Yaskawa INFORM job: SKRZYNIA_4740_90_STOPNI_20BR.JBI

/JOB
//NAME SKRZYNIA_4740_90_STOPNI_20BR
///FOLDERNAME 02-SKRZYNIE_JOBS
//POS
///NPOS 536,536,0,37,0,0
///TOOL 0
///POSTYPE PULSE
///PULSE
C00000=0,-52280,40443,0,6876,0
C00001=82314,-24956,17040,59626,-27382,6248
C00002=93910,-8625,17040,59626,-43355,6248
C00003=98846,-1061,-42166,80308,-57081,-16120
C00004=100452,6057,-48127,85711,-56704,-21322
C00005=95573,33077,-33257,84645,-64023,-26851
C00006=94102,33899,-31937,85246,-63371,-26689
C00007=95573,33077,-33257,84645,-64023,-26851
C00008=94862,31071,-36438,85313,-63677,-27192
C00009=95573,33077,-33257,84645,-64023,-26851
C00010=95263,33142,-33256,84677,-63995,-26850
C00011=95263,33142,-33256,84677,-63995,-26850
C00012=94017,33843,-32133,85187,-63445,-26710
C00013=95263,33142,-33256,84677,-63995,-26850
C00014=94657,31439,-35966,85248,-63701,-27141
C00015=95263,33142,-33256,84677,-63995,-26850
C00016=95260,33144,-33256,84678,-63995,-26850
C00017=95260,33144,-33256,84678,-63995,-26850
C00018=94022,33838,-32141,85183,-63448,-26711
C00019=95260,33144,-33256,84678,-63995,-26850
C00020=94618,31343,-36117,85281,-63684,-27157
C00021=95260,33144,-33256,84678,-63995,-26850
C00022=95258,25631,32269,66559,-75499,-2416
C00023=95258,25631,32269,66559,-75499,-2416
C00024=94181,26497,33533,66410,-74896,-2191
C00025=95658,30184,39035,66708,-78559,-2356
C00026=95217,30377,39331,66881,-79841,-2558
C00027=95258,25631,32269,66559,-75499,-2416
C00028=98811,21047,-15512,99242,-81394,-20987
C00029=98811,21047,-15512,99242,-81394,-20987
C00030=97775,21639,-14693,99563,-80753,-20993
C00031=98811,21047,-15512,99242,-81394,-20987
C00032=98206,18840,-18520,99489,-81124,-21211
C00033=98811,21047,-15512,99242,-81394,-20987
C00034=97770,33535,58109,97477,-73223,-2907
C00035=97471,32489,56434,97533,-73096,-3098
C00036=96615,33295,57725,97337,-72490,-3014
C00037=97471,32489,56434,97533,-73096,-3098
C00038=97097,30483,53272,97662,-72975,-3435
C00039=97471,32489,56434,97533,-73096,-3098
C00040=98003,23984,26658,100907,-76471,-9645
C00041=97707,-10819,-23052,107304,-59718,-16318
C00042=94212,-35028,-34485,100444,-49148,-11285
C00043=48287,-44591,-17414,16172,-14532,25809
C00044=85348,-13130,13838,41209,-47455,8220
C00045=97395,20012,29210,69700,-74457,-9077
C00046=97055,28839,36684,71776,-79389,-10554
C00047=97055,28839,36684,71776,-79389,-10554
C00048=96058,29646,37897,71666,-78799,-10362
C00049=97055,28839,36684,71776,-79389,-10554
C00050=96570,26659,33451,71832,-78911,-10777
C00051=97055,28839,36684,71776,-79389,-10554
C00052=99260,22658,16753,92099,-78835,-1091
C00053=98782,22427,16945,92082,-78485,-960
C00054=98098,22870,17565,92116,-78014,-935
C00055=98782,22427,16945,92082,-78485,-960
C00056=98488,21195,15235,92147,-78307,-1085
C00057=98782,22427,16945,92082,-78485,-960
C00058=99953,7972,-32104,116782,-84999,-13620
C00059=94704,-17776,-58548,118507,-81680,-13914
C00060=60067,-64368,-72505,144806,-26050,-19168
C00061=60067,-50244,-32501,110603,-14199,-2207
C00062=63330,-26972,24478,18707,-56801,31483
C00063=95462,-31003,-33042,65414,-41305,6524
C00064=97787,-9790,-26685,81509,-54738,-4408
C00065=99864,21793,7359,80466,-76601,-6182
C00066=99753,21489,3165,89598,-79157,-3178
C00067=99071,20978,1948,89791,-78725,-3400
C00068=98206,21502,2669,89926,-78149,-3364
C00069=99071,20978,1948,89791,-78725,-3400
C00070=98727,19613,87,89895,-78511,-3524
C00071=99071,20978,1948,89791,-78725,-3400
C00072=99862,21793,7358,80466,-76600,-6182
C00073=98290,21024,6297,80683,-75539,-6194
C00074=97471,21541,7008,80756,-75007,-6115
C00075=98290,21024,6297,80683,-75539,-6194
C00076=97834,19245,3873,80814,-75197,-6333
C00077=98290,21024,6297,80683,-75539,-6194
C00078=98946,26804,31705,85784,-78857,-1423
C00079=98946,26804,31705,85784,-78857,-1423
C00080=98292,27270,32391,85749,-78414,-1361
C00081=98946,26804,31705,85784,-78857,-1423
C00082=98631,25349,29587,85839,-78632,-1590
C00083=98946,26804,31705,85784,-78857,-1423
C00084=94295,-1388,2615,87521,-55608,-1527
C00085=77022,-27457,-20499,75297,-20933,3764
///LIMIT ON
C00086=42754,-66126,12236,-1301,3231,7194
///LIMIT OFF
C00087=0,-52280,40443,0,6876,0
C00088=0,-52280,40443,0,6876,0
C00089=50509,-19000,10610,51503,-15997,-61182
C00090=50873,-17966,11417,52677,-16048,-61710
C00091=49459,-16590,12517,51258,-15158,-61190
C00092=50592,-16429,12648,53120,-15720,-61960
C00093=50873,-17966,11417,52677,-16048,-61710
C00094=50703,-18403,11066,52155,-16024,-61477
C00095=50703,-18403,11066,52155,-16024,-61477
C00096=49026,-16768,12358,50435,-14971,-60844
C00097=50653,-16371,12680,53228,-15754,-62008
C00098=50703,-18403,11066,52155,-16024,-61477
C00099=50704,-18401,11069,52157,-16021,-61478
C00100=50704,-20525,5414,58956,-14779,-64789
C00101=49025,-18889,6668,57745,-13658,-64384
C00102=50799,-18420,7036,60610,-14610,-65581
C00103=50704,-20525,5414,58956,-14779,-64789
C00104=51005,-17995,11387,52847,-16122,-61778
C00105=51005,-17995,11387,52847,-16122,-61778
C00106=49564,-16598,12501,51417,-15218,-61257
C00107=50954,-16306,12737,53719,-15902,-62212
C00108=51005,-17995,11387,52847,-16122,-61778
C00109=51030,-17981,11395,52891,-16138,-61796
C00110=51030,-17981,11395,52891,-16138,-61796
C00111=49401,-16396,12662,51265,-15114,-61201
C00112=50908,-16047,12947,53789,-15850,-62250
C00113=51030,-17981,11395,52891,-16138,-61796
C00114=50945,-18019,11363,52741,-16103,-61737
C00115=50945,-16980,14081,49884,-16761,-60338
C00116=49117,-15186,15539,47848,-15653,-59576
C00117=50939,-14679,15960,50992,-16487,-60881
C00118=50945,-18019,11363,52741,-16103,-61737
C00119=50945,-18019,11363,52741,-16103,-61737
C00120=50945,-18556,9943,54337,-15776,-62517
C00121=48967,-16606,11493,52445,-14510,-61829
C00122=51083,-15952,12027,56053,-15559,-63336
C00123=50945,-18556,9943,54337,-15776,-62517
C00124=50945,-18019,11363,52741,-16103,-61737
C00125=51350,-15183,18375,46705,-17991,-58719
C00126=49319,-13187,20053,44263,-16830,-57796
C00127=51236,-12618,20544,47529,-17647,-59142
C00128=51350,-15183,18375,46705,-17991,-58719
C00129=50028,-23690,-6096,22921,-31075,-54538
C00130=50670,-23735,-6923,24003,-30760,-55076
C00131=48518,-21492,-5254,21861,-29696,-54082
C00132=50138,-21068,-4928,23831,-30039,-55022
C00133=50670,-23735,-6923,24003,-30760,-55076
C00134=49763,-24225,-29961,22080,-30065,-59113
C00135=49763,-24225,-29961,22080,-30065,-59113
C00136=47727,-21550,-27874,20313,-29013,-58119
C00137=49271,-21042,-27466,22016,-29310,-59069
C00138=49763,-24225,-29961,22080,-30065,-59113
C00139=50713,-12366,-58367,41124,-17813,-74400
C00140=50713,-12366,-58367,41124,-17813,-74400
C00141=48934,-9522,-55687,39981,-16902,-73526
C00142=50242,-8975,-55157,41389,-17374,-74448
C00143=50713,-12366,-58367,41124,-17813,-74400
C00144=50713,-12366,-58367,41124,-17813,-74400
C00145=50713,-12366,-58367,41124,-17813,-74400
C00146=48934,-9522,-55687,39981,-16902,-73526
C00147=50242,-8975,-55157,41389,-17374,-74448
C00148=50713,-12366,-58367,41124,-17813,-74400
C00149=49763,-25421,-36239,24565,-26935,-60445
C00150=43547,-31626,-19626,5157,-49140,-52118
C00151=40154,-51179,-915,24203,-8234,-36524
C00152=0,-52280,40443,0,6876,0
C00153=0,-52280,40443,0,6876,0
C00154=2117,-50103,-33543,4117,45077,-85249
C00155=-26439,-48928,-33543,4117,-52362,-85249
C00156=-1453,-29933,-32011,46693,-66666,-90474
C00157=24798,-19255,-10490,69050,-85424,-90395
C00158=18386,-22028,-12683,68302,-81515,-89477
///LIMIT ON
C00159=9843,-31743,-57176,61611,-65235,-99401
C00160=-39603,-23393,-71448,91573,-31907,-107123
C00161=-35705,5077,-63140,100511,-35979,-118164
C00162=-33789,12193,-59259,102607,-37482,-119984
C00163=-34998,13124,-58049,103267,-36945,-119997
C00164=-34401,14597,-56112,102586,-37131,-119778
C00165=-34998,13124,-58049,103267,-36945,-119997
C00166=-36388,13885,-57049,104079,-36338,-120048
C00167=-34998,13124,-58049,103267,-36945,-119997
C00168=-34008,-7969,-75285,118537,-50852,-116988
C00169=-26318,8527,-57077,128458,-81874,-108613
///LIMIT OFF
C00170=-23139,-1795,-12064,73373,-53703,-87448
C00171=-27830,-667,-10848,73187,-50621,-86997
C00172=-27373,916,-9115,73207,-50922,-87041
C00173=-27830,-667,-10848,73187,-50621,-86997
C00174=-28901,-207,-10348,73132,-49918,-86888
C00175=-27830,-667,-10848,73187,-50621,-86997
C00176=-37166,8347,13175,41366,-53536,-76331
C00177=-37403,7707,12401,41298,-53388,-76282
C00178=-36830,9273,14303,41455,-53750,-76396
C00179=-37403,7707,12401,41298,-53388,-76282
C00180=-38235,8246,13056,40951,-53040,-76025
C00181=-37403,7707,12401,41298,-53388,-76282
C00182=-30063,5992,18551,55847,-56234,-77619
C00183=-30754,7414,19761,55747,-55713,-77591
C00184=-30376,8670,21285,55817,-55984,-77619
C00185=-30754,7414,19761,55747,-55713,-77591
C00186=-31265,7672,20073,55566,-55435,-77478
C00187=-30085,6037,18588,55845,-56218,-77619
C00188=-25385,-1715,-9470,94765,-53990,-89712
C00189=-25885,-764,-8323,94779,-53645,-89697
C00190=-25564,418,-7032,94741,-53861,-89683
C00191=-25885,-764,-8323,94779,-53645,-89697
C00192=-26741,-428,-7957,94890,-53068,-89741
C00193=-25421,-1648,-9389,94767,-53966,-89710
C00194=-17789,-39335,-40320,90232,-41783,-86178
C00195=-25885,-761,-8324,94780,-53645,-89696
C00196=-25885,-761,-8324,94780,-53645,-89696
C00197=-25612,239,-7230,94748,-53828,-89684
C00198=-25885,-761,-8324,94780,-53645,-89696
C00199=-26712,-436,-7972,94885,-53087,-89742
C00200=-25885,-761,-8324,94780,-53645,-89696
C00201=-26038,-1317,-8919,94796,-53541,-89701
C00202=-18430,-29121,-33898,93348,-44706,-88207
C00203=-3209,-48313,-44409,84985,-37126,-83197
C00204=-3617,-53456,-46461,81793,-37023,-81323
C00205=-28991,-22310,-29554,94749,-46554,-89251
C00206=-30664,-6343,-14094,96248,-45630,-90223
C00207=-30664,-6343,-14094,96248,-45630,-90223
C00208=-30207,-5031,-12762,96238,-45949,-90236
C00209=-30664,-6343,-14094,96248,-45630,-90223
C00210=-31510,-5971,-13720,96406,-45066,-90297
C00211=-29506,-9179,-17232,96085,-46411,-90159
C00212=-30003,-8487,-16482,96169,-46079,-90194
C00213=-30881,-6301,-14053,96286,-45485,-90239
C00214=-30407,-4956,-12684,96275,-45813,-90252
C00215=-30881,-6301,-14053,96286,-45485,-90239
C00216=-31646,-5963,-13712,96429,-44974,-90305
C00217=-29893,-8752,-16772,96152,-46152,-90188
C00218=-30350,-7636,-15544,96220,-45845,-90215
C00219=-30881,-6301,-14053,96286,-45485,-90239
C00220=-30396,-4924,-12652,96275,-45822,-90251
C00221=-30881,-6301,-14053,96286,-45485,-90239
C00222=-31665,-5954,-13703,96434,-44961,-90308
C00223=-29959,-8593,-16598,96162,-46108,-90192
C00224=-26558,-19284,-27675,95285,-48332,-89713
C00225=-5136,-57382,-50746,80999,-31115,-81799
C00226=-5136,-57382,-50746,80999,-31115,-81799
C00227=-22762,-12288,-20025,94001,-55646,-89200
C00228=-24763,-3131,-11201,94769,-54426,-89746
C00229=-26203,-419,-7954,94818,-53430,-89712
C00230=-25939,548,-6896,94784,-53609,-89698
C00231=-26203,-419,-7954,94818,-53430,-89712
C00232=-26818,-174,-7689,94897,-53016,-89744
C00233=-24998,-2701,-10694,94780,-54264,-89743
C00234=-23275,-722,28392,94611,-50650,-77911
C00235=-21733,-16242,25206,75334,-39210,-63099
C00236=0,-52280,40443,0,6876,0
C00237=0,-52280,40443,0,6876,0
C00238=82314,-24956,17040,59626,-27382,6248
C00239=93910,-8625,17040,59626,-43355,6248
C00240=98846,-1061,-42166,80308,-57081,-16120
C00241=100452,6057,-48127,85711,-56704,-21322
C00242=95564,34698,-34234,85516,-63941,-27819
C00243=93687,36612,-31081,84292,-64733,-27467
C00244=93711,36598,-31105,84282,-64744,-27471
C00245=95564,34698,-34234,85516,-63941,-27819
C00246=95564,34698,-34234,85516,-63941,-27819
C00247=93687,36612,-31081,84292,-64733,-27467
C00248=93711,36598,-31105,84282,-64744,-27471
C00249=95564,34698,-34234,85516,-63941,-27819
C00250=96930,32282,-32252,82595,-65816,-26305
C00251=93663,32611,-31732,84127,-64318,-26195
C00252=93663,32611,-31732,84127,-64318,-26195
C00253=96930,32282,-32252,82595,-65816,-26305
C00254=96528,-7533,-34932,76119,-53878,-10439
C00255=88377,-34186,-45291,67238,-52212,-2442
C00256=73560,-62084,7826,28695,-34737,3666
C00257=0,-52280,40443,0,6876,0
C00258=0,-52280,40443,0,6876,0
C00259=2117,-50103,-33543,4117,45077,-85249
C00260=-26439,-48928,-33543,4117,-52362,-85249
C00261=-26439,-27355,-33543,41485,-52362,-85249
C00262=-39218,-24492,-41653,51934,-39374,-86964
C00263=-37997,-10433,-19136,70610,-34172,-88069
C00264=-38397,-8978,-17736,70703,-33874,-88109
C00265=-39218,-24492,-41653,51934,-39374,-86964
C00266=-26439,-27355,-33543,41485,-52362,-85249
C00267=1598,-24403,-16502,45671,-72599,-88798
C00268=-11365,-15171,10010,30164,-77975,-82960
C00269=-38112,4197,-14374,43778,-42973,-90436
C00270=-39116,7904,-10019,43942,-43580,-90646
C00271=-38495,8531,-9262,44482,-44499,-91194
C00272=-38112,4197,-14374,43778,-42973,-90436
C00273=-53220,-12364,-8957,19277,-47766,-73858
C00274=-11365,-15171,10010,30164,-77975,-82960
C00275=-16156,-38280,11293,23671,-42998,-42040
C00276=-11365,-47379,10010,30164,3063,-681
C00277=0,-52280,40443,0,6876,0
C00278=0,-36700,24612,-42871,-31823,-33862
C00279=44403,-30110,7154,24155,-23805,-45557
C00280=51347,-17798,16373,37641,-23556,-51399
C00281=51570,-17239,16856,38066,-23574,-51584
C00282=66153,-16343,3873,86567,-32078,-80939
C00283=60867,-15143,12446,70239,-26750,-71065
C00284=40431,-28773,9158,17648,-23273,-42875
C00285=0,-36700,24612,-42871,-31823,-33862
C00286=0,-52280,40443,0,6876,0
C00287=0,-52280,40443,0,6876,0
C00288=73560,-62084,7826,28695,-34737,3666
C00289=88377,-34186,-45291,67238,-52212,-2442
C00290=96920,-4461,-29697,76917,-56550,-10069
C00291=100432,21324,12575,83706,-77956,-7498
C00292=100432,21324,12575,83706,-77956,-7498
C00293=97224,21170,12361,83970,-75786,-7447
C00294=97224,21170,12361,83970,-75786,-7447
C00295=100432,21324,12575,83706,-77956,-7498
C00296=100432,21324,12575,83706,-77956,-7498
C00297=97481,25108,17890,83512,-78432,-7131
C00298=97624,25049,17805,83504,-78528,-7141
C00299=100432,21324,12575,83706,-77956,-7498
C00300=97137,1790,-11103,86179,-63102,-7963
C00301=99183,2264,5333,86781,-62651,-3264
C00302=99868,-33,22146,72719,-59601,5126
C00303=99028,-10516,17309,71061,-60695,4227
C00304=58820,-39124,10926,53325,-41870,3759
C00305=0,-52280,40443,0,6876,0
C00306=37281,-50778,-9546,79570,-75313,-71156
C00307=21038,-23698,-30323,82948,-81132,-85647
C00308=-27256,-5882,-14331,85818,-48304,-85968
C00309=-24751,2890,-4920,85349,-55822,-86178
C00310=-24793,2953,-4845,85351,-55796,-86173
C00311=-27256,-5882,-14331,85818,-48304,-85968
C00312=-21143,-15675,-23596,84785,-52496,-85466
C00313=35274,-15248,-23220,82440,-90817,-86704
C00314=35274,-15248,-23220,82440,-90817,-86704
C00315=-45551,161,-18089,35087,-36064,-73293
C00316=-42435,6767,-10562,40540,-41185,-77662
C00317=-42821,6494,-10882,40094,-40673,-77276
C00318=-45551,161,-18089,35087,-36064,-73293
C00319=-32891,-7184,-22739,69075,-41395,-83248
C00320=-29265,-39765,-39402,58096,-43152,-73226
C00321=-37287,-55159,35520,2191,5667,-2084
C00322=0,-52280,40443,0,6876,0
C00323=0,-52280,40443,0,6876,0
C00324=0,-52280,40443,0,6876,0
C00325=73560,-62084,7826,28695,-34737,3666
C00326=96983,-27116,-23481,78724,-62297,-1998
C00327=100467,-7393,-15195,81625,-60158,-6002
C00328=99336,18440,8642,84276,-74234,-7647
C00329=99336,18440,8642,84276,-74234,-7647
C00330=97735,24994,14595,85350,-78994,-5109
C00331=97744,25074,13580,86004,-79195,-4385
C00332=99336,18440,8642,84276,-74234,-7647
C00333=98746,26047,40390,96212,-73340,-2686
C00334=96511,23274,36200,96292,-71976,-3182
C00335=96511,27155,48340,94664,-71177,-571
C00336=99747,18296,13811,99163,-76345,-8478
C00337=99017,774,-48740,120026,-82763,-23886
C00338=82685,-42461,-85506,125714,-59125,-24709
///LIMIT ON
C00339=37721,-67612,11381,1325,-438,7850
///LIMIT OFF
C00340=-37287,-55159,35520,2191,5667,-2084
C00341=-40042,-68802,-18337,47708,-19461,-45384
C00342=-28646,-23138,-32952,89786,-42552,-85395
C00343=-38882,-16596,-17625,44304,-41043,-72768
C00344=-42680,-6319,-12818,46127,-36112,-73823
C00345=-37459,704,-5408,52536,-43357,-78192
C00346=-32778,4349,-7465,59128,-48375,-83352
C00347=-42680,-6319,-12818,46127,-36112,-73823
C00348=-38882,-16596,-17625,44304,-41043,-72768
C00349=-28646,-23138,-32952,89786,-42552,-85395
C00350=-29905,-15291,-26411,91102,-43435,-86304
C00351=-25469,1350,-9790,89991,-54827,-86555
C00352=-24242,3379,-7505,89554,-57286,-86471
C00353=-29905,-15291,-26411,91102,-43435,-86304
C00354=-40042,-68802,-18337,47708,-19461,-45384
C00355=-37287,-55159,35520,2191,5667,-2084
C00356=0,-52280,40443,0,6876,0
C00357=37164,-60659,6466,13301,-5027,-19773
C00358=45362,-39990,2831,27538,-17767,-40935
C00359=57189,-26834,-7130,38780,-31731,-51561
C00360=63456,-14144,8594,45591,-40850,-50620
C00361=63445,-23884,-40761,66084,-30994,-63296
C00362=57189,-26834,-7130,38780,-31731,-51561
C00363=41180,-61187,4729,17280,-8498,-23442
C00364=0,-52280,40443,0,6876,0
C00365=0,-52280,40443,0,6876,0
///LIMIT ON
C00366=37721,-67612,11381,1325,-438,7850
///LIMIT OFF
C00367=43180,-50572,-20637,6552,-29302,38834
C00368=69362,-40002,-13521,39754,-33332,24421
C00369=86483,-21864,2840,55410,-40116,17549
C00370=99420,-11049,13736,67201,-51390,13904
C00371=92855,-5018,12828,77373,-48606,10660
C00372=98199,21452,7696,88481,-78015,-298
C00373=98177,26799,35147,85763,-78047,6724
C00374=100920,18905,27694,85174,-73370,7184
C00375=94483,-7610,-22783,94358,-54968,-958
C00376=98124,-17779,-18471,95902,-51295,3087
C00377=88943,-29687,-12397,76321,-42166,11919
C00378=82008,-39290,-17962,63915,-40768,19941
C00379=-36913,-32963,-979,75363,-26772,-58744
C00380=-42264,1508,8544,35869,-47237,-69477
C00381=-43183,4597,12058,35318,-46938,-69128
C00382=-43183,5775,16318,34276,-48598,-68388
C00383=-42264,1508,8544,35869,-47237,-69477
C00384=56258,-38103,3288,28818,-33580,-23051
C00385=41438,-37635,17580,13151,-29920,-38779
C00386=54964,-26842,8528,44141,-23181,-52038
C00387=50761,-21373,7883,46957,-18149,-54038
C00388=65129,-17418,-4929,103101,-32265,-89308
C00389=65181,-6263,27418,81207,-31059,-77222
C00390=56762,-20631,11812,69834,-24329,-69917
C00391=46096,-45842,-2681,20981,-19497,-36310
C00392=41180,-61187,4729,17280,-8498,-23442
C00393=0,-52280,40443,0,6876,0
C00394=0,-52280,40443,0,6876,0
///LIMIT ON
C00395=37721,-67612,11381,1325,-438,7850
///LIMIT OFF
C00396=43180,-50572,-20637,6552,-29302,38834
C00397=79425,-37128,-15462,51820,-35721,18807
C00398=92377,-29666,-26166,73570,-38078,7008
C00399=97441,-6012,-18634,86114,-58345,-2339
C00400=98864,-2001,-14672,90389,-62789,-3799
C00401=98767,21176,13691,87588,-77304,-2577
C00402=98123,23617,17097,87345,-78645,-2335
C00403=97979,23711,17231,87352,-78549,-2326
C00404=98864,-2001,-14672,90389,-62789,-3799
C00405=100472,-329,-13432,98539,-67097,-6304
C00406=92822,-26306,-37175,103295,-43881,-7703
C00407=68601,-52593,-52127,95725,-25602,-3235
C00408=80632,-38079,-20908,64053,-45216,12949
C00409=43180,-50572,-20637,6552,-29302,38834
///LIMIT ON
C00410=37721,-67612,11381,1325,-438,7850
///LIMIT OFF
C00411=0,-52280,40443,0,6876,0
C00412=0,-52280,40443,0,6876,0
C00413=0,-52280,40443,0,-39412,36675
C00414=-54026,-30203,28811,-7745,-28969,-5087
C00415=-30389,-9386,-5824,79667,-43789,-73484
C00416=-32979,-3325,255,79720,-41988,-73575
C00417=-25304,6223,10893,81656,-55729,-74481
C00418=-23842,8927,14147,81883,-58875,-74544
C00419=-30389,-9386,-5824,79667,-43789,-73484
C00420=-32145,-6440,-2937,79673,-42575,-73527
C00421=-25014,6414,11121,81706,-56254,-74506
C00422=-23603,11547,23533,79434,-59735,-72187
C00423=-32145,-5050,2357,77009,-42992,-71800
C00424=-35251,-18143,20376,53513,-41117,-59413
C00425=-9534,-43450,13514,26959,-29486,-38723
C00426=-22834,-59963,22946,6692,-2150,-9612
C00427=0,-52280,40443,0,6876,0
///LIMIT ON
C00428=23708,-46776,23536,16027,-4787,-19738
///LIMIT OFF
C00429=50917,-40459,4132,34421,-18173,-42391
C00430=51059,-36587,4608,36647,-19418,-45358
C00431=50113,-22729,10834,36393,-23396,-50963
C00432=62046,-17757,4067,79440,-27252,-76630
C00433=63763,-15682,7486,80006,-29481,-77057
C00434=50113,-22729,10834,36393,-23396,-50963
C00435=31287,-69981,-10850,7253,-6843,-20996
C00436=19644,-57271,30737,863,5243,-2499
C00437=0,-52280,40443,0,6876,0
C00438=0,-52280,40443,0,6876,0
C00439=37721,-67612,11381,1325,-438,7850
C00440=43180,-50572,-20637,6552,-29302,38834
C00441=79425,-37128,-15462,51820,-35721,18807
C00442=92377,-33385,-41303,83059,-36844,1354
C00443=97441,-6012,-18634,86114,-58345,-2339
C00444=98442,-3149,-15680,86092,-59018,-2413
C00445=97114,-5888,-18685,94010,-59218,-3940
C00446=99563,18710,13338,88899,-76218,-2010
C00447=98011,23070,19863,88505,-78125,-1416
C00448=98011,24865,28095,87725,-78063,621
C00449=100205,15202,-8793,101167,-79304,-9541
C00450=100471,12680,2182,89317,-73847,-3746
C00451=93923,-8883,-21959,92925,-54783,-4609
C00452=92822,-26306,-37175,103295,-43881,-7703
C00453=68601,-52593,-52127,95725,-25602,-3235
C00454=80632,-38079,-20908,64053,-45216,12949
C00455=43180,-50572,-20637,6552,-29302,38834
C00456=37721,-67612,11381,1325,-438,7850
C00457=0,-52280,40443,0,6876,0
C00458=0,-52280,40443,0,6876,0
C00459=0,-52280,40443,0,-39412,36675
C00460=-54026,-30203,28811,-7745,-28969,-5087
C00461=-81492,-18979,22896,-11682,-23662,-26316
C00462=-32145,-2720,10458,73217,-43826,-69319
C00463=-32145,-2720,10458,73217,-43826,-69319
C00464=-25800,12961,35355,74076,-56913,-68018
C00465=-23961,12723,28512,77913,-59573,-70804
C00466=-32145,-2720,10458,73217,-43826,-69319
C00467=-34274,-9754,-24316,117159,-46217,-86271
C00468=-34274,-9754,-24316,117159,-46217,-86271
C00469=-29822,-1437,-15851,112752,-53901,-84078
C00470=-28945,-336,-14662,112011,-55335,-83695
C00471=-34274,-9754,-24316,117159,-46217,-86271
C00472=-34422,-9999,20796,72411,-42519,-66994
C00473=-35251,-18143,20376,53513,-41117,-59413
C00474=-9534,-43450,13514,26959,-29486,-38723
C00475=-22834,-59963,22946,6692,-2150,-9612
C00476=0,-52280,40443,0,6876,0
C00477=29449,-70637,-48792,-22650,-13229,-23678
C00478=49121,-28282,-35458,21895,-29219,-59001
C00479=50484,-13386,-55713,36158,-19724,-71897
C00480=55938,-10187,-55661,55618,-22248,-82832
C00481=57381,15206,-57369,78100,-21009,-89969
C00482=50484,-13386,-55713,36158,-19724,-71897
C00483=49763,-25421,-36239,24565,-26935,-60445
C00484=50529,-22709,-3778,22940,-31995,-54502
C00485=45389,-28224,4312,35967,-15579,-54278
C00486=40154,-51179,-915,24203,-8234,-36524
C00487=0,-52280,40443,0,6876,0
C00488=0,-52280,40443,0,6876,0
///LIMIT ON
C00489=37721,-67612,11381,1325,-438,7850
///LIMIT OFF
C00490=43181,-50571,-20637,6551,-29300,38834
C00491=92325,-23846,-7228,63960,-40898,12897
C00492=85232,-2754,25377,50981,-49542,17626
C00493=95618,10017,30418,66150,-65403,10402
C00494=98328,26728,37723,75385,-78922,5377
C00495=99185,24817,27312,82025,-78466,1195
C00496=97766,23970,26102,82043,-77480,1145
C00497=97755,21890,16078,83086,-77017,-1370
C00498=100993,19573,16602,81480,-76704,-137
C00499=97988,24882,21615,85608,-78767,-653
C00500=97988,24882,21615,85608,-78767,-653
C00501=97883,29022,44703,72741,-79810,7156
C00502=99525,21729,17159,85870,-76787,-954
C00503=97991,25479,22462,85564,-79108,-597
C00504=97991,25479,22462,85564,-79108,-597
C00505=99525,21729,17159,85870,-76787,-954
C00506=99525,21703,17016,85886,-76785,-991
C00507=98063,26874,26717,84040,-79605,457
C00508=97834,25035,16764,84912,-79171,-2109
C00509=100039,22069,12584,85154,-78124,-2393
C00510=100072,10223,-2816,88932,-70713,-3891
C00511=99051,-8427,5223,77933,-54888,7183
C00512=82477,-27884,-1524,62699,-44420,15528
C00513=0,-52278,40443,0,6872,5
C00514=0,-52278,40443,31822,-65283,-46097
C00515=-7820,3000,44222,77356,-66876,-70486
C00516=-24244,23423,72059,64993,-61079,-67138
C00517=-27261,30732,84230,62108,-60720,-65392
C00518=-22394,37028,87531,68934,-68535,-64461
C00519=-24244,23423,72059,64993,-61079,-67138
C00520=3014,-20441,-7349,104591,-68614,-79454
C00521=6322,-14118,13197,96169,-69167,-72790
C00522=14133,-16757,18528,88010,-59455,-67296
C00523=-10261,-46634,14475,36899,-22136,-31570
C00524=-22834,-59963,22946,6692,-2150,-9612
C00525=0,-52280,40443,0,6876,0
///LIMIT ON
C00526=23708,-46776,23536,16027,-4787,-19738
///LIMIT OFF
C00527=50917,-40459,4132,34421,-18173,-42391
C00528=49876,-21948,7530,68838,-10324,-59148
C00529=46721,-18942,9765,68167,-8197,-59205
C00530=59504,-15355,-1382,118573,-27610,-87938
C00531=59094,-13899,7128,105147,-23854,-78064
C00532=45927,-22803,4403,78462,-8511,-64553
C00533=62498,-35400,-2607,72048,-19281,-59202
C00534=31287,-69981,-10850,7253,-6843,-20996
C00535=0,-52280,40443,0,6876,0
BC00000=502871
BC00001=460491
BC00002=460491
BC00003=460491
BC00004=460491
BC00005=483588
BC00006=483588
BC00007=483588
BC00008=483588
BC00009=483588
BC00010=529782
BC00011=529782
BC00012=529782
BC00013=529782
BC00014=529782
BC00015=529782
BC00016=575949
BC00017=575949
BC00018=575949
BC00019=575949
BC00020=575949
BC00021=575949
BC00022=551765
BC00023=551765
BC00024=551765
BC00025=551765
BC00026=551765
BC00027=551765
BC00028=597819
BC00029=597819
BC00030=597819
BC00031=597819
BC00032=597819
BC00033=597819
BC00034=565028
BC00035=565028
BC00036=565028
BC00037=565028
BC00038=565028
BC00039=565028
BC00040=565028
BC00041=565028
BC00042=548653
BC00043=714482
BC00044=729478
BC00045=787852
BC00046=785759
BC00047=785759
BC00048=785759
BC00049=785759
BC00050=785759
BC00051=785759
BC00052=818809
BC00053=818809
BC00054=818809
BC00055=818809
BC00056=818809
BC00057=818809
BC00058=820354
BC00059=820354
BC00060=872244
BC00061=872244
BC00062=844509
BC00063=938343
BC00064=932297
BC00065=935100
BC00066=888948
BC00067=888948
BC00068=888948
BC00069=888948
BC00070=888948
BC00071=888948
BC00072=933770
BC00073=933770
BC00074=933770
BC00075=933770
BC00076=933770
BC00077=933770
BC00078=933164
BC00079=933164
BC00080=933164
BC00081=933164
BC00082=933164
BC00083=933164
BC00084=915220
BC00085=922555
BC00086=827037
BC00087=781071
BC00088=781071
BC00089=857334
BC00090=903417
BC00091=903417
BC00092=903417
BC00093=903417
BC00094=846075
BC00095=846075
BC00096=846075
BC00097=846075
BC00098=846075
BC00099=780190
BC00100=780190
BC00101=780190
BC00102=780190
BC00103=780190
BC00104=722535
BC00105=722535
BC00106=722535
BC00107=722535
BC00108=722535
BC00109=657432
BC00110=657432
BC00111=657432
BC00112=657432
BC00113=657432
BC00114=600107
BC00115=600107
BC00116=600107
BC00117=600107
BC00118=600107
BC00119=534593
BC00120=534593
BC00121=534593
BC00122=534593
BC00123=534593
BC00124=477174
BC00125=477174
BC00126=477174
BC00127=477174
BC00128=477174
BC00129=474905
BC00130=474905
BC00131=474905
BC00132=474905
BC00133=474905
BC00134=474905
BC00135=474905
BC00136=474905
BC00137=474905
BC00138=474905
BC00139=474905
BC00140=474905
BC00141=474905
BC00142=474905
BC00143=474905
BC00144=428822
BC00145=428822
BC00146=428822
BC00147=428822
BC00148=428822
BC00149=474905
BC00150=477686
BC00151=548577
BC00152=548577
BC00153=492150
BC00154=423885
BC00155=423885
BC00156=519103
BC00157=542802
BC00158=634915
BC00159=493160
BC00160=493160
BC00161=517936
BC00162=517447
BC00163=516208
BC00164=516208
BC00165=516208
BC00166=516208
BC00167=516208
BC00168=525487
BC00169=485388
BC00170=500803
BC00171=500803
BC00172=500803
BC00173=500803
BC00174=500803
BC00175=500803
BC00176=585253
BC00177=585253
BC00178=585253
BC00179=585253
BC00180=585253
BC00181=585253
BC00182=600589
BC00183=600589
BC00184=600589
BC00185=600589
BC00186=600589
BC00187=600589
BC00188=646713
BC00189=646713
BC00190=646713
BC00191=646713
BC00192=646713
BC00193=646713
BC00194=659006
BC00195=692822
BC00196=692822
BC00197=692822
BC00198=692822
BC00199=692822
BC00200=692822
BC00201=669701
BC00202=669701
BC00203=669701
BC00204=791136
BC00205=762000
BC00206=762000
BC00207=762000
BC00208=762000
BC00209=762000
BC00210=762000
BC00211=762000
BC00212=831025
BC00213=831025
BC00214=831025
BC00215=831025
BC00216=831025
BC00217=831025
BC00218=877128
BC00219=877128
BC00220=877128
BC00221=877128
BC00222=877128
BC00223=877128
BC00224=854090
BC00225=854090
BC00226=990684
BC00227=992363
BC00228=992364
BC00229=992364
BC00230=992364
BC00231=992364
BC00232=992364
BC00233=992364
BC00234=941750
BC00235=932032
BC00236=798985
BC00237=460491
BC00238=460491
BC00239=460491
BC00240=460491
BC00241=460491
BC00242=445216
BC00243=445216
BC00244=437592
BC00245=445216
BC00246=491299
BC00247=491299
BC00248=483675
BC00249=491299
BC00250=530690
BC00251=530690
BC00252=523002
BC00253=530690
BC00254=557568
BC00255=557568
BC00256=557568
BC00257=557568
BC00258=492150
BC00259=423885
BC00260=423885
BC00261=423885
BC00262=423885
BC00263=406365
BC00264=406365
BC00265=423885
BC00266=423885
BC00267=423885
BC00268=423885
BC00269=507950
BC00270=507950
BC00271=500226
BC00272=507950
BC00273=493160
BC00274=493160
BC00275=493160
BC00276=493160
BC00277=493160
BC00278=598171
BC00279=670543
BC00280=727463
BC00281=728141
BC00282=728141
BC00283=784926
BC00284=789114
BC00285=598171
BC00286=508521
BC00287=557568
BC00288=557568
BC00289=557568
BC00290=600794
BC00291=559125
BC00292=474638
BC00293=474638
BC00294=467026
BC00295=474638
BC00296=536109
BC00297=536109
BC00298=543829
BC00299=536109
BC00300=524597
BC00301=582327
BC00302=566813
BC00303=561271
BC00304=584417
BC00305=584417
BC00306=542360
BC00307=521200
BC00308=474976
BC00309=474976
BC00310=482600
BC00311=474976
BC00312=474976
BC00313=474976
BC00314=630364
BC00315=628593
BC00316=624867
BC00317=617183
BC00318=631527
BC00319=617183
BC00320=617427
BC00321=620193
BC00322=620193
BC00323=542207
BC00324=542207
BC00325=542207
BC00326=541760
BC00327=590944
BC00328=571989
BC00329=582221
BC00330=582229
BC00331=589997
BC00332=582221
BC00333=573417
BC00334=573417
BC00335=573417
BC00336=573417
BC00337=592950
BC00338=619041
BC00339=665809
BC00340=620193
BC00341=620193
BC00342=635598
BC00343=635598
BC00344=635598
BC00345=635598
BC00346=635598
BC00347=635598
BC00348=635598
BC00349=635598
BC00350=658627
BC00351=658627
BC00352=666320
BC00353=658627
BC00354=620193
BC00355=620193
BC00356=620193
BC00357=576903
BC00358=514129
BC00359=467432
BC00360=467432
BC00361=467436
BC00362=467432
BC00363=539526
BC00364=539526
BC00365=748464
BC00366=748464
BC00367=748464
BC00368=661500
BC00369=661494
BC00370=661494
BC00371=661494
BC00372=694447
BC00373=678206
BC00374=678206
BC00375=699767
BC00376=699767
BC00377=675213
BC00378=655721
BC00379=696009
BC00380=735643
BC00381=735643
BC00382=739967
BC00383=735643
BC00384=632579
BC00385=598230
BC00386=596115
BC00387=604917
BC00388=604917
BC00389=642244
BC00390=649618
BC00391=551933
BC00392=576449
BC00393=563161
BC00394=748464
BC00395=748464
BC00396=748464
BC00397=748464
BC00398=748464
BC00399=748464
BC00400=755892
BC00401=755892
BC00402=755892
BC00403=763572
BC00404=755892
BC00405=765830
BC00406=765830
BC00407=765830
BC00408=798734
BC00409=810658
BC00410=748464
BC00411=748464
BC00412=672709
BC00413=672709
BC00414=762701
BC00415=743900
BC00416=736524
BC00417=736351
BC00418=743900
BC00419=743900
BC00420=759331
BC00421=759331
BC00422=759331
BC00423=759331
BC00424=750104
BC00425=672725
BC00426=672725
BC00427=672725
BC00428=782243
BC00429=806462
BC00430=818228
BC00431=851878
BC00432=851878
BC00433=910395
BC00434=851878
BC00435=618402
BC00436=618402
BC00437=618402
BC00438=733103
BC00439=733103
BC00440=748464
BC00441=748464
BC00442=748464
BC00443=748464
BC00444=831044
BC00445=819602
BC00446=818299
BC00447=818299
BC00448=818299
BC00449=818299
BC00450=802063
BC00451=801971
BC00452=735108
BC00453=735108
BC00454=783373
BC00455=795297
BC00456=733103
BC00457=733103
BC00458=672709
BC00459=672709
BC00460=762701
BC00461=791880
BC00462=819491
BC00463=819491
BC00464=817331
BC00465=817331
BC00466=817326
BC00467=863478
BC00468=863478
BC00469=863478
BC00470=871062
BC00471=863478
BC00472=774095
BC00473=750104
BC00474=672725
BC00475=672725
BC00476=672725
BC00477=543617
BC00478=474905
BC00479=474905
BC00480=474905
BC00481=451867
BC00482=474905
BC00483=474905
BC00484=474905
BC00485=474901
BC00486=548577
BC00487=548577
BC00488=748464
BC00489=748464
BC00490=914315
BC00491=907949
BC00492=897350
BC00493=904390
BC00494=916313
BC00495=879003
BC00496=879003
BC00497=879003
BC00498=878712
BC00499=947035
BC00500=954731
BC00501=916313
BC00502=939340
BC00503=939340
BC00504=947006
BC00505=939340
BC00506=901871
BC00507=901871
BC00508=901871
BC00509=901871
BC00510=907639
BC00511=880549
BC00512=861365
BC00513=762878
BC00514=921533
BC00515=958534
BC00516=946591
BC00517=946591
BC00518=946592
BC00519=954904
BC00520=963295
BC00521=934184
BC00522=908449
BC00523=754884
BC00524=672725
BC00525=672725
BC00526=577701
BC00527=467723
BC00528=467723
BC00529=467723
BC00530=467723
BC00531=528577
BC00532=527471
BC00533=527369
BC00534=757643
BC00535=757643
///POSTYPE BASE
///RECTAN
///RCONF 1,0,0,0,0,0,0,0,0,0,0,0,0,0,0,0,0,0,0,0,0,0,0,0
P00006=0.000,0.000,0.000,0.0000,0.0000,0.0000
///RCONF 0,0,0,0,0,0,0,0,0,0,0,0,0,0,0,0,0,0,0,0,0,0,0,0
P00058=0.000,0.000,3.000,0.0000,0.0000,0.0000
///RCONF 1,0,0,0,0,0,0,0,0,0,0,0,0,0,0,0,0,0,0,0,0,0,0,0
P00300=-0.036,-1.505,2.318,0.0000,0.0000,0.0000
P00301=0.046,-2.112,7.779,0.0000,0.0000,0.0000
P00302=-0.180,-2.409,6.326,0.0000,0.0000,0.0000
///RCONF 0,0,0,0,0,0,0,0,0,0,0,0,0,0,0,0,0,0,0,0,0,0,0,0
P00303=-0.004,-1.437,-4.584,0.0000,0.0000,0.0000
P00304=0.028,-1.666,-4.234,0.0000,0.0000,0.0000
P00305=-0.003,-1.920,-3.501,0.0000,0.0000,0.0000
P00307=0.019,-2.151,-5.077,0.0000,0.0000,0.0000
P00308=-0.003,-2.092,-4.888,0.0000,0.0000,0.0000
P00309=-0.040,-2.205,-4.992,0.0000,0.0000,0.0000
P00310=-0.006,-2.490,-5.925,0.0000,0.0000,0.0000
P00311=-0.007,-2.079,-5.307,0.0000,0.0000,0.0000
P00351=13.563,-0.027,-0.653,0.0000,0.0000,0.0000
P00352=13.252,-0.027,-0.827,0.0000,0.0000,0.0000
P00353=10.971,-0.082,0.776,0.0000,0.0000,0.0000
P00354=-0.024,2.508,-1.824,0.0000,0.0000,0.0000
P00355=-0.001,2.528,-1.131,0.0000,0.0000,0.0000
P00356=-0.034,2.921,-0.262,0.0000,0.0000,0.0000
P00357=0.003,3.386,-0.091,0.0000,0.0000,0.0000
P00358=0.014,3.037,-0.020,0.0000,0.0000,0.0000
P00359=-0.005,2.731,0.912,0.0000,0.0000,0.0000
P00360=-0.011,3.412,0.438,0.0000,0.0000,0.0000
P00361=0.018,3.050,1.253,0.0000,0.0000,0.0000
P00362=0.014,2.784,0.148,0.0000,0.0000,0.0000
P00400=5.920,-3.503,-0.024,0.0000,0.0000,0.0000
P00401=3.430,-0.021,1.131,0.0000,0.0000,0.0000
P00402=-0.253,1.107,3.062,0.0000,0.0000,0.0000
P00403=-3.666,-0.015,5.328,0.0000,0.0000,0.0000
///RCONF 1,0,0,0,0,0,0,0,0,0,0,0,0,0,0,0,0,0,0,0,0,0,0,0
P00404=0.029,4.189,-1.030,0.0000,0.0000,0.0000
///RCONF 0,0,0,0,0,0,0,0,0,0,0,0,0,0,0,0,0,0,0,0,0,0,0,0
P00405=2.420,0.007,1.427,0.0000,0.0000,0.0000
P00406=3.513,-0.022,0.429,0.0000,0.0000,0.0000
///RCONF 1,0,0,0,1,0,0,0,0,0,0,0,0,0,0,0,0,0,0,0,0,0,0,0
P00407=-0.029,2.348,-1.469,0.0000,0.0000,0.0000
P00408=0.010,1.346,-1.479,0.0000,0.0000,0.0000
///RCONF 1,0,0,0,0,0,0,0,0,0,0,0,0,0,0,0,0,0,0,0,0,0,0,0
P00409=-0.026,2.090,-1.483,0.0000,0.0000,0.0000
P00410=0.001,4.491,-0.583,0.0000,0.0000,0.0000
///RCONF 1,0,0,0,1,0,0,0,0,0,0,0,0,0,0,0,0,0,0,0,0,0,0,0
P00411=-0.015,3.627,0.872,0.0000,0.0000,0.0000
//INST
///DATE 2025/02/06 12:50
///ATTR SC,RW
///GROUP1 RB1,BS1
NOP
CALL JOB:MOVE_INTO_TUNNEL
MOVJ C00000 BC00000 VJ=10.00
MOVJ C00001 BC00001 VJ=30.00
MOVJ C00002 BC00002 VJ=30.00
MOVL C00003 BC00003 V=500.0
MOVJ C00004 BC00004 VJ=30.00
'------------------------
'W65.3
'------------------------
MOVL C00005 BC00005 V=333.3 PL=0
REFP 3 C00006 BC00006
CALL JOB:SEARCH-R1
SET P0300 P0006
SFTON P0300
MOVL C00007 BC00007 V=333.3 PL=0
REFP 3 C00008 BC00008
CALL JOB:SEARCH-R1
SET P0300 P0006
SFTON P0300
MOVL C00009 BC00009 V=333.3 PL=0
SFTOF
'------------------------
'W65.5
'------------------------
MOVL C00010 BC00010 V=500.0
MOVL C00011 BC00011 V=333.3 PL=0
REFP 3 C00012 BC00012
CALL JOB:SEARCH-R1
SET P0301 P0006
SFTON P0301
MOVL C00013 BC00013 V=333.3 PL=0
REFP 3 C00014 BC00014
CALL JOB:SEARCH-R1
SET P0301 P0006
SFTON P0301
MOVL C00015 BC00015 V=333.3 PL=0
SFTOF
'------------------------
'W65.7
'------------------------
MOVL C00016 BC00016 V=500.0
MOVL C00017 BC00017 V=333.3 PL=0
REFP 3 C00018 BC00018
CALL JOB:SEARCH-R1
SET P0302 P0006
SFTON P0302
MOVL C00019 BC00019 V=333.3 PL=0
REFP 3 C00020 BC00020
CALL JOB:SEARCH-R1
SET P0302 P0006
SFTON P0302
MOVL C00021 BC00021 V=500.0 PL=0
SFTOF
'------------------------
'W65.10
'------------------------
MOVL C00022 BC00022 V=500.0
MOVL C00023 BC00023 V=333.3 PL=0
REFP 3 C00024 BC00024
CALL JOB:SEARCH-R1
SET P0303 P0006
SFTON P0303
MOVL C00025 BC00025 V=333.3 PL=0
REFP 3 C00026 BC00026
CALL JOB:SEARCH-R1
SET P0303 P0006
SFTON P0303
MOVL C00027 BC00027 V=333.3 PL=0
SFTOF
'------------------------
'W65.12
'------------------------
MOVL C00028 BC00028 V=500.0
MOVL C00029 BC00029 V=333.3 PL=0
REFP 3 C00030 BC00030
CALL JOB:SEARCH-R1
SET P0304 P0006
SFTON P0304
MOVL C00031 BC00031 V=333.3 PL=0
REFP 3 C00032 BC00032
CALL JOB:SEARCH-R1
SET P0304 P0006
SFTON P0304
MOVL C00033 BC00033 V=333.3 PL=0
SFTOF
'------------------------
'W65.15
'------------------------
MOVL C00034 BC00034 V=500.0
MOVL C00035 BC00035 V=333.3 PL=0
REFP 3 C00036 BC00036
CALL JOB:SEARCH-R1
SET P0305 P0006
SFTON P0305
MOVL C00037 BC00037 V=333.3 PL=0
REFP 3 C00038 BC00038
CALL JOB:SEARCH-R1
SET P0305 P0006
SFTON P0305
MOVL C00039 BC00039 V=333.3 PL=0
SFTOF
'------------------------
'W65.17
'------------------------
MOVL C00040 BC00040 V=500.0
MOVL C00041 BC00041 V=333.3
MOVL C00042 BC00042 V=500.0
MOVJ C00043 BC00043 VJ=30.00
MOVL C00044 BC00044 V=500.0
MOVL C00045 BC00045 V=500.0
'------------------------
'W65.20
'------------------------
MOVL C00046 BC00046 V=500.0
MOVL C00047 BC00047 V=333.3 PL=0
REFP 3 C00048 BC00048
CALL JOB:SEARCH-R1
SET P0307 P0006
SFTON P0307
MOVL C00049 BC00049 V=333.3 PL=0
REFP 3 C00050 BC00050
CALL JOB:SEARCH-R1
SET P0307 P0006
SFTON P0307
MOVL C00051 BC00051 V=500.0 PL=0
SFTOF
'------------------------
'W65.23
'------------------------
MOVL C00052 BC00052 V=500.0
MOVL C00053 BC00053 V=333.3 PL=0
REFP 3 C00054 BC00054
CALL JOB:SEARCH-R1
SET P0308 P0006
SFTON P0308
MOVL C00055 BC00055 V=333.3 PL=0
REFP 3 C00056 BC00056
CALL JOB:SEARCH-R1
SET P0308 P0006
SFTON P0308
MOVL C00057 BC00057 V=500.0 PL=0
SFTOF
'------------------------
'W65.25
'------------------------
MOVL C00058 BC00058 V=333.3
MOVL C00059 BC00059 V=333.3
MOVL C00060 BC00060 V=500.0
MOVL C00061 BC00061 V=500.0
MOVL C00062 BC00062 V=250.0
MOVL C00063 BC00063 V=500.0
MOVL C00064 BC00064 V=500.0
MOVL C00065 BC00065 V=83.3
MOVL C00066 BC00066 V=500.0
MOVL C00067 BC00067 V=333.3 PL=0
REFP 3 C00068 BC00068
CALL JOB:SEARCH-R1
SET P0309 P0006
SFTON P0309
MOVL C00069 BC00069 V=333.3 PL=0
REFP 3 C00070 BC00070
CALL JOB:SEARCH-R1
SET P0309 P0006
SFTON P0309
MOVL C00071 BC00071 V=500.0 PL=0
SFTOF
'------------------------
'W65.28
'------------------------
MOVL C00072 BC00072 V=500.0
MOVL C00073 BC00073 V=333.3 PL=0
REFP 3 C00074 BC00074
CALL JOB:SEARCH-R1
SET P0310 P0006
SFTON P0310
MOVL C00075 BC00075 V=333.3 PL=0
REFP 3 C00076 BC00076
CALL JOB:SEARCH-R1
SET P0310 P0006
SFTON P0310
MOVL C00077 BC00077 V=333.3 PL=0
SFTOF
'------------------------
'W65.30
'------------------------
MOVL C00078 BC00078 V=500.0
MOVL C00079 BC00079 V=333.3 PL=0
REFP 3 C00080 BC00080
CALL JOB:SEARCH-R1
SET P0311 P0006
SFTON P0311
MOVL C00081 BC00081 V=333.3 PL=0
REFP 3 C00082 BC00082
CALL JOB:SEARCH-R1
SET P0311 P0006
SFTON P0311
MOVL C00083 BC00083 V=333.3 PL=0
SFTOF
MOVL C00084 BC00084 V=500.0
MOVL C00085 BC00085 V=500.0
MOVJ C00086 BC00086 VJ=30.00
MOVJ C00087 BC00087 VJ=30.00
MOVJ C00088 BC00088 VJ=30.00
'------------------------
MOVJ C00089 BC00089 VJ=30.00
MOVL C00090 BC00090 V=333.3 PL=0
REFP 3 C00091 BC00091
CALL JOB:SEARCH-R1
IMOV P0058 V=16.7
SET P0351 P0006
SFTON P0351
REFP 3 C00092 BC00092
CALL JOB:SEARCH-R1
SET P0351 P0006
SFTON P0351
MOVL C00093 BC00093 V=500.0 PL=0
SFTOF
'------------------------
'W254A L
'------------------------
MOVJ C00094 BC00094 VJ=30.00
MOVL C00095 BC00095 V=333.3 PL=0
REFP 3 C00096 BC00096
CALL JOB:SEARCH-R1
IMOV P0058 V=16.7
SET P0352 P0006
SFTON P0352
REFP 3 C00097 BC00097
CALL JOB:SEARCH-R1
SET P0352 P0006
SFTON P0352
MOVL C00098 BC00098 V=500.0 PL=0
SFTOF
'------------------------
'W250A P
'------------------------
MOVJ C00099 BC00099 VJ=30.00
MOVL C00100 BC00100 V=333.3 PL=0
REFP 3 C00101 BC00101
CALL JOB:SEARCH-R1
IMOV P0058 V=16.7
SET P0353 P0006
SFTON P0353
REFP 3 C00102 BC00102
CALL JOB:SEARCH-R1
SET P0353 P0006
SFTON P0353
MOVL C00103 BC00103 V=500.0 PL=0
SFTOF
'------------------------
'W250A L
'------------------------
MOVJ C00104 BC00104 VJ=30.00
MOVL C00105 BC00105 V=333.3 PL=0
REFP 3 C00106 BC00106
CALL JOB:SEARCH-R1
IMOV P0058 V=16.7
SET P0354 P0006
SFTON P0354
REFP 3 C00107 BC00107
CALL JOB:SEARCH-R1
SET P0354 P0006
SFTON P0354
MOVL C00108 BC00108 V=500.0 PL=0
SFTOF
'------------------------
'W253A P
'------------------------
MOVJ C00109 BC00109 VJ=30.00
MOVL C00110 BC00110 V=333.3 PL=0
REFP 3 C00111 BC00111
CALL JOB:SEARCH-R1
IMOV P0058 V=16.7
SET P0355 P0006
SFTON P0355
REFP 3 C00112 BC00112
CALL JOB:SEARCH-R1
SET P0355 P0006
SFTON P0355
MOVL C00113 BC00113 V=333.3 PL=0
SFTOF
'------------------------
'W253A L
'------------------------
MOVJ C00114 BC00114 VJ=30.00
MOVL C00115 BC00115 V=333.3 PL=0
REFP 3 C00116 BC00116
CALL JOB:SEARCH-R1
IMOV P0058 V=16.7
SET P0356 P0006
SFTON P0356
REFP 3 C00117 BC00117
CALL JOB:SEARCH-R1
SET P0356 P0006
SFTON P0356
MOVL C00118 BC00118 V=500.0 PL=0
SFTOF
'------------------------
'W256A P
'------------------------
MOVJ C00119 BC00119 VJ=30.00
MOVL C00120 BC00120 V=333.3 PL=0
REFP 3 C00121 BC00121
CALL JOB:SEARCH-R1
IMOV P0058 V=16.7
SET P0357 P0006
SFTON P0357
REFP 3 C00122 BC00122
CALL JOB:SEARCH-R1
SET P0357 P0006
SFTON P0357
MOVL C00123 BC00123 V=500.0 PL=0
SFTOF
'------------------------
'W256A L
'------------------------
MOVJ C00124 BC00124 VJ=30.00
MOVL C00125 BC00125 V=333.3 PL=0
REFP 3 C00126 BC00126
CALL JOB:SEARCH-R1
IMOV P0058 V=16.7
SET P0358 P0006
SFTON P0358
REFP 3 C00127 BC00127
CALL JOB:SEARCH-R1
SET P0358 P0006
SFTON P0358
MOVL C00128 BC00128 V=500.0 PL=0
SFTOF
'------------------------
'W252A P
'------------------------
MOVL C00129 BC00129 V=500.0
MOVL C00130 BC00130 V=333.3 PL=0
REFP 3 C00131 BC00131
CALL JOB:SEARCH-R1
IMOV P0058 V=16.7
SET P0359 P0006
SFTON P0359
REFP 3 C00132 BC00132
CALL JOB:SEARCH-R1
SET P0359 P0006
SFTON P0359
MOVL C00133 BC00133 V=333.3 PL=0
SFTOF
'------------------------
'W252A L
'------------------------
MOVL C00134 BC00134 V=500.0
MOVL C00135 BC00135 V=333.3 PL=0
REFP 3 C00136 BC00136
CALL JOB:SEARCH-R1
IMOV P0058 V=16.7
SET P0360 P0006
SFTON P0360
REFP 3 C00137 BC00137
CALL JOB:SEARCH-R1
SET P0360 P0006
SFTON P0360
MOVL C00138 BC00138 V=500.0 PL=0
SFTOF
'------------------------
'W255A
'------------------------
MOVL C00139 BC00139 V=500.0
MOVL C00140 BC00140 V=333.3 PL=0
REFP 3 C00141 BC00141
CALL JOB:SEARCH-R1
IMOV P0058 V=16.7
SET P0361 P0006
SFTON P0361
REFP 3 C00142 BC00142
CALL JOB:SEARCH-R1
SET P0361 P0006
SFTON P0361
MOVL C00143 BC00143 V=500.0 PL=0
SFTOF
MOVL C00144 BC00144 V=500.0
MOVL C00145 BC00145 V=333.3 PL=0
REFP 3 C00146 BC00146
CALL JOB:SEARCH-R1
IMOV P0058 V=16.7
SET P0362 P0006
SFTON P0362
REFP 3 C00147 BC00147
CALL JOB:SEARCH-R1
SET P0361 P0006
SFTON P0362
MOVL C00148 BC00148 V=500.0 PL=0
SFTOF
MOVL C00149 BC00149 V=500.0
MOVJ C00150 BC00150 VJ=50.00
MOVJ C00151 BC00151 VJ=50.00
MOVJ C00152 BC00152 VJ=50.00
COMM MOVJ C00153 BC00153 VJ=30.00
COMM MOVJ C00154 BC00154 VJ=30.00
COMM MOVJ C00155 BC00155 VJ=30.00
COMM MOVJ C00156 BC00156 VJ=50.00
COMM 'COMMENT
COMM MOVJ C00157 BC00157 VJ=50.00
COMM MOVJ C00158 BC00158 VJ=30.00
COMM GETE D040 P0400 (1)
COMM GETE D041 P0400 (2)
COMM GETE D042 P0400 (3)
COMM SETE P0401 (1) D040
COMM SETE P0401 (2) D041
COMM SETE P0401 (3) D042
COMM GETE D040 P0400 (1)
COMM GETE D041 P0400 (2)
COMM GETE D042 P0400 (3)
COMM SETE P0402 (1) D040
COMM SETE P0402 (2) D041
COMM SETE P0402 (3) D042
COMM MOVL C00159 BC00159 V=333.3
COMM MOVL C00160 BC00160 V=333.3
COMM MOVL C00161 BC00161 V=333.3
COMM MOVL C00162 BC00162 V=333.3
COMM '------------------------
COMM 'W61.5
COMM '------------------------
COMM MOVL C00163 BC00163 V=66.7 PL=0
COMM REFP 3 C00164 BC00164
COMM CALL JOB:SEARCH-R1
COMM SET P0401 P0006
COMM SFTON P0401
COMM MOVL C00165 BC00165 V=66.7 PL=0
COMM REFP 3 C00166 BC00166
COMM CALL JOB:SEARCH-R1
COMM SET P0401 P0006
COMM SFTON P0401
COMM MOVL C00167 BC00167 V=66.7 PL=0
COMM SFTOF
COMM MOVL C00168 BC00168 V=333.3
COMM MOVL C00169 BC00169 V=333.3
COMM '------------------------
COMM 'W61.7
COMM '------------------------
COMM MOVL C00170 BC00170 V=333.3
COMM MOVL C00171 BC00171 V=66.7 PL=0
COMM REFP 3 C00172 BC00172
COMM CALL JOB:SEARCH-R1
COMM SET P0402 P0006
COMM SFTON P0402
COMM MOVL C00173 BC00173 V=66.7 PL=0
COMM REFP 3 C00174 BC00174
COMM CALL JOB:SEARCH-R1
COMM SET P0402 P0006
COMM SFTON P0402
COMM MOVL C00175 BC00175 V=66.7 PL=0
COMM SFTOF
COMM '------------------------
COMM 'W61.10
COMM '------------------------
COMM MOVL C00176 BC00176 V=500.0
COMM MOVL C00177 BC00177 V=166.7 PL=0
COMM REFP 3 C00178 BC00178
COMM CALL JOB:SEARCH-R1
COMM SET P0403 P0006
COMM SFTON P0403
COMM MOVL C00179 BC00179 V=166.7 PL=0
COMM REFP 3 C00180 BC00180
COMM CALL JOB:SEARCH-R1
COMM SET P0403 P0006
COMM SFTON P0403
COMM MOVL C00181 BC00181 V=500.0 PL=0
COMM SFTOF
COMM '------------------------
COMM 'W61.12
COMM '------------------------
COMM MOVL C00182 BC00182 V=500.0
COMM MOVL C00183 BC00183 V=166.7 PL=0
COMM REFP 3 C00184 BC00184
COMM CALL JOB:SEARCH-R1
COMM SET P0404 P0006
COMM SFTON P0404
COMM MOVL C00185 BC00185 V=166.7 PL=0
COMM REFP 3 C00186 BC00186
COMM CALL JOB:SEARCH-R1
COMM SET P0404 P0006
COMM SFTON P0404
COMM MOVL C00187 BC00187 V=500.0 PL=0
COMM SFTOF
COMM '------------------------
COMM 'W61.15
COMM '------------------------
COMM MOVL C00188 BC00188 V=500.0
COMM MOVL C00189 BC00189 V=166.7 PL=0
COMM REFP 3 C00190 BC00190
COMM CALL JOB:SEARCH-R1
COMM SET P0405 P0006
COMM SFTON P0405
COMM MOVL C00191 BC00191 V=166.7 PL=0
COMM REFP 3 C00192 BC00192
COMM CALL JOB:SEARCH-R1
COMM SET P0405 P0006
COMM SFTON P0405
COMM MOVL C00193 BC00193 V=500.0 PL=0
COMM SFTOF
COMM MOVL C00194 BC00194 V=500.0
COMM SFTOF
COMM GETE D040 P0405 (1)
COMM GETE D041 P0405 (2)
COMM GETE D042 P0405 (3)
COMM SETE P0406 (1) D040
COMM SETE P0406 (2) D041
COMM SETE P0406 (3) D042
COMM '------------------------
COMM 'W61.17
COMM '------------------------
COMM MOVL C00195 BC00195 V=333.3
COMM MOVL C00196 BC00196 V=66.7 PL=0
COMM REFP 3 C00197 BC00197
COMM CALL JOB:SEARCH-R1
COMM SET P0406 P0006
COMM SFTON P0406
COMM MOVL C00198 BC00198 V=66.7 PL=0
COMM REFP 3 C00199 BC00199
COMM CALL JOB:SEARCH-R1
COMM SET P0406 P0006
COMM SFTON P0406
COMM MOVL C00200 BC00200 V=66.7 PL=0
COMM SFTOF
COMM MOVL C00201 BC00201 V=333.3
COMM MOVL C00202 BC00202 V=333.3
COMM MOVJ C00203 BC00203 VJ=30.00
COMM MOVJ C00204 BC00204 VJ=50.00
COMM MOVL C00205 BC00205 V=666.7
COMM '------------------------
COMM 'W61.20
COMM '------------------------
COMM MOVL C00206 BC00206 V=500.0
COMM MOVL C00207 BC00207 V=166.7 PL=0
COMM REFP 3 C00208 BC00208
COMM CALL JOB:SEARCH-R1
COMM SET P0407 P0006
COMM SFTON P0407
COMM MOVL C00209 BC00209 V=166.7 PL=0
COMM REFP 3 C00210 BC00210
COMM CALL JOB:SEARCH-R1
COMM SET P0407 P0006
COMM SFTON P0407
COMM MOVL C00211 BC00211 V=500.0 PL=0
COMM SFTOF
COMM '------------------------
COMM 'W61.23
COMM '------------------------
COMM MOVL C00212 BC00212 V=500.0
COMM MOVL C00213 BC00213 V=166.7 PL=0
COMM REFP 3 C00214 BC00214
COMM CALL JOB:SEARCH-R1
COMM SET P0408 P0006
COMM SFTON P0408
COMM MOVL C00215 BC00215 V=166.7 PL=0
COMM REFP 3 C00216 BC00216
COMM CALL JOB:SEARCH-R1
COMM SET P0408 P0006
COMM SFTON P0408
COMM MOVL C00217 BC00217 V=500.0 PL=0
COMM SFTOF
COMM '------------------------
COMM 'W61.25
COMM '------------------------
COMM MOVL C00218 BC00218 V=500.0
COMM MOVL C00219 BC00219 V=166.7 PL=0
COMM REFP 3 C00220 BC00220
COMM CALL JOB:SEARCH-R1
COMM SET P0409 P0006
COMM SFTON P0409
COMM MOVL C00221 BC00221 V=166.7 PL=0
COMM REFP 3 C00222 BC00222
COMM CALL JOB:SEARCH-R1
COMM SET P0409 P0006
COMM SFTON P0409
COMM MOVL C00223 BC00223 V=500.0 PL=0
COMM SFTOF
COMM MOVL C00224 BC00224 V=500.0
COMM MOVL C00225 BC00225 V=500.0
COMM MOVJ C00226 BC00226 VJ=50.00
COMM MOVL C00227 BC00227 V=666.7
COMM GETE D040 P0409 (1)
COMM GETE D041 P0409 (2)
COMM GETE D042 P0409 (3)
COMM SETE P0410 (1) D040
COMM SETE P0410 (2) D041
COMM SETE P0410 (3) D042
COMM '------------------------
COMM 'W61.30
COMM '------------------------
COMM MOVL C00228 BC00228 V=500.0
COMM MOVL C00229 BC00229 V=166.7 PL=0
COMM REFP 3 C00230 BC00230
COMM CALL JOB:SEARCH-R1
COMM SET P0411 P0006
COMM SFTON P0411
COMM MOVL C00231 BC00231 V=166.7 PL=0
COMM REFP 3 C00232 BC00232
COMM CALL JOB:SEARCH-R1
COMM SET P0411 P0006
COMM SFTON P0411
COMM MOVL C00233 BC00233 V=500.0 PL=0
COMM SFTOF
COMM MOVL C00234 BC00234 V=666.7
COMM MOVJ C00235 BC00235 VJ=30.00
MOVJ C00236 BC00236 VJ=50.00
CALL JOB:FRONT_SEARCH_90ST-2_4740
MOVJ C00237 BC00237 VJ=50.00
MOVJ C00238 BC00238 VJ=40.00
MOVJ C00239 BC00239 VJ=30.00
MOVL C00240 BC00240 V=666.7
MOVJ C00241 BC00241 VJ=40.00
'------------------------
'W65.3
'------------------------
SFTON P0300
MOVL C00242 BC00242 V=500.0
MOVL C00243 BC00243 V=333.3 PL=0
MACRO1 MJ#(0) ARGF10
ARCON
MOVL C00244 BC00244 V=10.8
ARCOF
MOVL C00245 BC00245 V=166.7
MOVL C00246 BC00246 V=500.0
MOVL C00247 BC00247 V=333.3 PL=0
MACRO1 MJ#(0) ARGF10
ARCON
MOVL C00248 BC00248 V=10.8
ARCOF
MOVL C00249 BC00249 V=166.7
SFTOF
'------------------------
'W65.5
'------------------------
SFTON P0301
MOVL C00250 BC00250 V=333.3
MOVL C00251 BC00251 V=133.3 PL=0
MACRO1 MJ#(0) ARGF10
ARCON
MOVL C00252 BC00252 V=10.8
ARCOF
MOVL C00253 BC00253 V=166.7
SFTOF
MOVL C00254 BC00254 V=500.0
MOVL C00255 BC00255 V=333.3
MOVJ C00256 BC00256 VJ=25.00
MOVJ C00257 BC00257 VJ=50.00
'::::::::::::::::::::::::::::::::
'::::::::::::::::::::::::::::::::
'::::::::::::::::::::::::::::::::
'::::::::::::::::::::::::::::::::
'::::::::::::::::::::::::::::::::
COMM MOVJ C00258 BC00258 VJ=50.00
COMM MOVJ C00259 BC00259 VJ=50.00
COMM MOVJ C00260 BC00260 VJ=50.00
COMM MOVJ C00261 BC00261 VJ=50.00
COMM MOVJ C00262 BC00262 VJ=20.00
COMM '------------------------
COMM 'W61.3
COMM '------------------------
COMM SFTON P0400
COMM MOVL C00263 BC00263 V=333.3
COMM MOVL C00264 BC00264 V=66.7 PL=0
COMM MACRO1 MJ#(0) ARGF9
COMM ARCOF
COMM SFTOF
COMM 'BELKA PRZEJAZD
COMM MOVJ C00265 BC00265 VJ=25.00
COMM MOVJ C00266 BC00266 VJ=50.00
COMM MOVL C00267 BC00267 V=500.0
COMM MOVL C00268 BC00268 V=500.0
COMM '------------------------
COMM 'W61.5
COMM '------------------------
COMM SFTON P0401
COMM MOVL C00269 BC00269 V=333.3
COMM MOVL C00270 BC00270 V=133.3 PL=0
COMM MACRO1 MJ#(0) ARGF24
COMM ARCON
COMM MOVL C00271 BC00271 V=7.5
COMM ARCOF
COMM MOVL C00272 BC00272 V=250.0
COMM SFTOF
COMM MOVL C00273 BC00273 V=333.3
COMM MOVJ C00274 BC00274 VJ=35.00
COMM MOVJ C00275 BC00275 VJ=50.00
COMM MOVJ C00276 BC00276 VJ=50.00
COMM MOVJ C00277 BC00277 VJ=50.00
MOVJ C00278 BC00278 VJ=50.00
MOVJ C00279 BC00279 VJ=50.00
MOVJ C00280 BC00280 VJ=50.00
'------------------------
'W250A
'------------------------
SFTON P0354
MOVL C00281 BC00281 V=333.3
MOVL C00282 BC00282 V=133.3 PL=0
MACRO1 MJ#(0) ARGF29
ARCON
SFTOF
SFTON P0353
MOVL C00283 BC00283 V=12.5
ARCOF
MOVL C00284 BC00284 V=166.7
SFTOF
MOVJ C00285 BC00285 VJ=50.00
MOVJ C00286 BC00286 VJ=50.00
MOVJ C00287 BC00287 VJ=50.00
MOVJ C00288 BC00288 VJ=50.00
MOVJ C00289 BC00289 VJ=50.00
MOVJ C00290 BC00290 VJ=20.00
MOVJ C00291 BC00291 VJ=10.00
'------------------------
'W65.7
'------------------------
SFTON P0302
'MOTOSIM PULSE LIMIT
MOVL C00292 BC00292 V=500.0
MOVL C00293 BC00293 V=133.3 PL=0
MACRO1 MJ#(0) ARGF30
ARCON
MOVL C00294 BC00294 V=11.7
ARCOF
MOVL C00295 BC00295 V=250.0
SFTOF
'------------------------
'W65.10
'------------------------
SFTON P0303
MOVL C00296 BC00296 V=500.0
MOVL C00297 BC00297 V=166.7 PL=0
ARCON
MOVL C00298 BC00298 V=11.7
ARCOF
MOVL C00299 BC00299 V=166.7
SFTOF
COMM SFTOF
COMM MOVL C00300 BC00300 V=333.3
COMM MOVL C00301 BC00301 V=500.0
COMM MOVJ C00302 BC00302 VJ=50.00
COMM MOVJ C00303 BC00303 VJ=30.00
COMM MOVJ C00304 BC00304 VJ=50.00
COMM MOVJ C00305 BC00305 VJ=50.00
COMM '::::::::::::::::::::::::::::::::
COMM '::::::::::::::::::::::::::::::::
COMM '------------------------
COMM 'W61.7
COMM '------------------------
COMM '::::::::::::::::::::::::::::::::
COMM '::::::::::::::::::::::::::::::::
COMM MOVJ C00306 BC00306 VJ=50.00
COMM MOVJ C00307 BC00307 VJ=35.00
COMM SFTON P0402
COMM MOVL C00308 BC00308 V=333.3
COMM MOVL C00309 BC00309 V=133.3 PL=0
COMM MACRO1 MJ#(0) ARGF24
COMM ARCON
COMM MOVL C00310 BC00310 V=7.5
COMM ARCOF
COMM MOVL C00311 BC00311 V=166.7
COMM SFTOF
COMM MOVL C00312 BC00312 V=500.0
COMM MOVL C00313 BC00313 V=500.0
COMM MOVJ C00314 BC00314 VJ=50.00
COMM '------------------------
COMM 'W61.10
COMM '------------------------
COMM SFTON P0403
COMM MOVL C00315 BC00315 V=333.3
COMM MOVL C00316 BC00316 V=133.3 PL=0
COMM MACRO1 MJ#(0) ARGF24
COMM ARCON
COMM MOVL C00317 BC00317 V=7.5
COMM ARCOF
COMM MOVL C00318 BC00318 V=166.7
COMM SFTOF
COMM MOVL C00319 BC00319 V=333.3
COMM MOVJ C00320 BC00320 VJ=35.00
COMM MOVJ C00321 BC00321 VJ=50.00
COMM MOVJ C00322 BC00322 VJ=50.00
COMM '::::::::::::::::::::::::
COMM '::::::::::::::::::::::::
COMM '::::::::::::::::::::::::
COMM '::::::::::::::::::::::::
COMM '::::::::::::::::::::::::
COMM '::::::::::::::::::::::::
COMM '::::::::::::::::::::::::
COMM MOVJ C00323 BC00323 VJ=50.00
COMM MOVJ C00324 BC00324 VJ=50.00
COMM MOVJ C00325 BC00325 VJ=50.00
COMM MOVJ C00326 BC00326 VJ=50.00
COMM MOVJ C00327 BC00327 VJ=50.00
COMM MOVJ C00328 BC00328 VJ=20.00
'------------------------
'W65.12
'------------------------
SFTON P0304
MOVL C00329 BC00329 V=333.3
MOVL C00330 BC00330 V=133.3 PL=0
MACRO1 MJ#(0) ARGF30
ARCON
MOVL C00331 BC00331 V=11.7
ARCOF
MOVL C00332 BC00332 V=166.7
SFTOF
'------------------------
'W65.15
'------------------------
SFTON P0305
MOVL C00333 BC00333 V=333.3
MOVL C00334 BC00334 V=166.7 PL=0
ARCON
MOVL C00335 BC00335 V=11.7
ARCOF
MOVL C00336 BC00336 V=166.7
SFTOF
MOVL C00337 BC00337 V=333.3
MOVL C00338 BC00338 V=500.0
MOVJ C00339 BC00339 VJ=50.00
COMM '::::::::::::::::::::::::
COMM '::::::::::::::::::::::::
COMM '::::::::::::::::::::::::
COMM '::::::::::::::::::::::::
COMM '::::::::::::::::::::::::
COMM '::::::::::::::::::::::::
COMM '::::::::::::::::::::::::
COMM MOVJ C00340 BC00340 VJ=50.00
COMM MOVJ C00341 BC00341 VJ=50.00
COMM '::::::::::::::::::::::::::::::::
COMM '::::::::::::::::::::::::::::::::
COMM '------------------------
COMM 'W61.12
COMM '------------------------
COMM '::::::::::::::::::::::::::::::::
COMM '::::::::::::::::::::::::::::::::
COMM SFTON P0404
COMM MOVJ C00342 BC00342 VJ=50.00
COMM MOVL C00343 BC00343 V=333.3
COMM MOVL C00344 BC00344 V=333.3
COMM MOVL C00345 BC00345 V=166.7 PL=0
COMM MACRO1 MJ#(0) ARGF24
COMM ARCON
COMM MOVL C00346 BC00346 V=7.5
COMM ARCOF
COMM MOVL C00347 BC00347 V=166.7
COMM SFTOF
COMM MOVL C00348 BC00348 V=333.3
COMM MOVL C00349 BC00349 V=333.3
COMM '------------------------
COMM 'W61.15
COMM '------------------------
COMM SFTON P0405
COMM MOVL C00350 BC00350 V=333.3
COMM MOVL C00351 BC00351 V=166.7 PL=0
COMM MACRO1 MJ#(0) ARGF24
COMM ARCON
COMM MOVL C00352 BC00352 V=7.5
COMM ARCOF
COMM MOVL C00353 BC00353 V=166.7
COMM SFTOF
COMM MOVJ C00354 BC00354 VJ=50.00
COMM MOVJ C00355 BC00355 VJ=50.00
COMM MOVJ C00356 BC00356 VJ=50.00
COMM '::::::::::::::::::::::::
COMM '::::::::::::::::::::::::
COMM '::::::::::::::::::::::::
COMM '::::::::::::::::::::::::
COMM '::::::::::::::::::::::::
COMM '::::::::::::::::::::::::
COMM '::::::::::::::::::::::::
MOVJ C00357 BC00357 VJ=50.00
MOVJ C00358 BC00358 VJ=50.00
'------------------------
'W252A
'------------------------
SFTON P0359
MOVL C00359 BC00359 V=500.0
MOVL C00360 BC00360 V=166.7 PL=0
MACRO1 MJ#(0) ARGF29
ARCON
SFTOF
SFTON P0358
MOVL C00361 BC00361 V=12.5
ARCOF
MOVL C00362 BC00362 V=250.0
SFTOF
MOVJ C00363 BC00363 VJ=50.00
MOVJ C00364 BC00364 VJ=80.00
MOVJ C00365 BC00365 VJ=80.00
MOVJ C00366 BC00366 VJ=50.00
MOVJ C00367 BC00367 VJ=50.00
MOVJ C00368 BC00368 VJ=25.00
MOVL C00369 BC00369 V=333.3
MOVL C00370 BC00370 V=333.3
'------------------------
'W65.17
'------------------------
MOVL C00371 BC00371 V=166.7
SFTON P0305
MOVL C00372 BC00372 V=166.7 PL=0
MACRO1 MJ#(0) ARGF30
ARCON
MOVL C00373 BC00373 V=11.7
ARCOF
SFTOF
MOVL C00374 BC00374 V=166.7
SFTOF
MOVL C00375 BC00375 V=250.0
MOVL C00376 BC00376 V=250.0
MOVL C00377 BC00377 V=333.3
MOVJ C00378 BC00378 VJ=25.00
'::::::::::::::::::::::::
'::::::::::::::::::::::::
'::::::::::::::::::::::::
'::::::::::::::::::::::::
'::::::::::::::::::::::::
'::::::::::::::::::::::::
'::::::::::::::::::::::::
'::::::::::::::::::::::::::::::::
'::::::::::::::::::::::::::::::::
'------------------------
'W61.17
'------------------------
'::::::::::::::::::::::::::::::::
'::::::::::::::::::::::::::::::::
COMM SFTON P0406
COMM MOVJ C00379 BC00379 VJ=10.00
COMM MOVL C00380 BC00380 V=150.0
COMM MOVL C00381 BC00381 V=66.7 PL=0
COMM MACRO1 MJ#(0) ARGF24
COMM ARCON
COMM MOVL C00382 BC00382 V=6.7
COMM ARCOF
COMM MOVL C00383 BC00383 V=83.3
COMM SFTOF
'------------------------
'W253A
'------------------------
MOVJ C00384 BC00384 VJ=50.00
MOVJ C00385 BC00385 VJ=50.00
SFTON P0356
MOVL C00386 BC00386 V=333.3
MOVL C00387 BC00387 V=333.3
MOVL C00388 BC00388 V=166.7 PL=0
MACRO1 MJ#(0) ARGF29
ARCON
SFTOF
SFTON P0355
MOVL C00389 BC00389 V=12.5
ARCOF
MOVL C00390 BC00390 V=250.0
SFTOF
MOVJ C00391 BC00391 VJ=50.00
MOVJ C00392 BC00392 VJ=50.00
MOVJ C00393 BC00393 VJ=80.00
MOVJ C00394 BC00394 VJ=80.00
MOVJ C00395 BC00395 VJ=50.00
MOVJ C00396 BC00396 VJ=50.00
MOVJ C00397 BC00397 VJ=50.00
MOVJ C00398 BC00398 VJ=30.00
MOVJ C00399 BC00399 VJ=30.00
'------------------------
'W65.20
'------------------------
SFTON P0307
MOVL C00400 BC00400 V=333.3
MOVL C00401 BC00401 V=166.7
MOVL C00402 BC00402 V=166.7 PL=0
MACRO1 MJ#(0) ARGF30
ARCON
MOVL C00403 BC00403 V=11.7
ARCOF
MOVL C00404 BC00404 V=250.0
SFTOF
MOVL C00405 BC00405 V=333.3
MOVL C00406 BC00406 V=333.3
MOVL C00407 BC00407 V=333.3
MOVJ C00408 BC00408 VJ=50.00
MOVJ C00409 BC00409 VJ=50.00
MOVJ C00410 BC00410 VJ=50.00
MOVJ C00411 BC00411 VJ=50.00
COMM '::::::::::::::::::::::::
COMM '::::::::::::::::::::::::
COMM '::::::::::::::::::::::::
COMM '::::::::::::::::::::::::
COMM '::::::::::::::::::::::::
COMM '::::::::::::::::::::::::
COMM '::::::::::::::::::::::::
COMM MOVJ C00412 BC00412 VJ=80.00
COMM MOVJ C00413 BC00413 VJ=50.00
COMM MOVJ C00414 BC00414 VJ=50.00
COMM '::::::::::::::::::::::::::::::::
COMM '::::::::::::::::::::::::::::::::
COMM '------------------------
COMM 'W61.20
COMM '------------------------
COMM '::::::::::::::::::::::::::::::::
COMM '::::::::::::::::::::::::::::::::
COMM SFTON P0407
COMM MOVL C00415 BC00415 V=333.3
COMM MOVL C00416 BC00416 V=166.7
COMM MOVL C00417 BC00417 V=133.3 PL=0
COMM MACRO1 MJ#(0) ARGF24
COMM ARCON
COMM MOVL C00418 BC00418 V=7.5
COMM ARCOF
COMM MOVL C00419 BC00419 V=166.7
COMM SFTOF
COMM SFTON P0407
COMM MOVL C00420 BC00420 V=166.7
COMM MOVL C00421 BC00421 V=133.3 PL=0
COMM MACRO1 MJ#(0) ARGF24
COMM ARCON
COMM MOVL C00422 BC00422 V=7.5
COMM ARCOF
COMM MOVL C00423 BC00423 V=166.7
COMM SFTOF
COMM '::::::::::::::::::::::::
COMM '::::::::::::::::::::::::
COMM '::::::::::::::::::::::::
COMM '::::::::::::::::::::::::
COMM '::::::::::::::::::::::::
COMM MOVJ C00424 BC00424 VJ=50.00
COMM MOVJ C00425 BC00425 VJ=50.00
COMM MOVJ C00426 BC00426 VJ=50.00
COMM MOVJ C00427 BC00427 VJ=50.00
COMM '------------------------
COMM 'W254A
COMM '------------------------
MOVJ C00428 BC00428 VJ=50.00
MOVJ C00429 BC00429 VJ=50.00
SFTON P0352
MOVL C00430 BC00430 V=500.0
MOVL C00431 BC00431 V=500.0
MOVL C00432 BC00432 V=166.7 PL=0
MACRO1 MJ#(0) ARGF29
ARCON
SFTOF
SFTON P0351
MOVL C00433 BC00433 V=12.5
ARCOF
MOVL C00434 BC00434 V=333.3
SFTOF
COMM MOVJ C00435 BC00435 VJ=80.00
COMM MOVJ C00436 BC00436 VJ=80.00
COMM MOVJ C00437 BC00437 VJ=80.00
COMM MOVJ C00438 BC00438 VJ=80.00
COMM MOVJ C00439 BC00439 VJ=50.00
MOVJ C00440 BC00440 VJ=50.00
MOVJ C00441 BC00441 VJ=50.00
MOVJ C00442 BC00442 VJ=50.00
MOVJ C00443 BC00443 VJ=30.00
MOVL C00444 BC00444 V=500.0
'------------------------
'W65.23
'------------------------
SFTON P0308
MOVL C00445 BC00445 V=333.3
MOVL C00446 BC00446 V=166.7
MOVL C00447 BC00447 V=133.3 PL=0
MACRO1 MJ#(0) ARGF30
ARCON
MOVL C00448 BC00448 V=11.7
ARCOF
MOVL C00449 BC00449 V=166.7
SFTOF
'------------------------
'W65.25
'------------------------
MOVL C00450 BC00450 V=500.0
MOVL C00451 BC00451 V=333.3
MOVL C00452 BC00452 V=500.0
MOVL C00453 BC00453 V=333.3
COMM MOVJ C00454 BC00454 VJ=50.00
COMM MOVJ C00455 BC00455 VJ=50.00
COMM MOVJ C00456 BC00456 VJ=50.00
COMM MOVJ C00457 BC00457 VJ=80.00
COMM '::::::::::::::::::::::::
COMM '::::::::::::::::::::::::
COMM '::::::::::::::::::::::::
COMM '::::::::::::::::::::::::
COMM '::::::::::::::::::::::::
COMM '::::::::::::::::::::::::
COMM '::::::::::::::::::::::::
COMM MOVJ C00458 BC00458 VJ=80.00
COMM MOVJ C00459 BC00459 VJ=80.00
COMM MOVJ C00460 BC00460 VJ=50.00
COMM MOVJ C00461 BC00461 VJ=50.00
COMM '::::::::::::::::::::::::::::::::
COMM '::::::::::::::::::::::::::::::::
COMM '------------------------
COMM 'W61.23
COMM '------------------------
COMM '::::::::::::::::::::::::::::::::
COMM '::::::::::::::::::::::::::::::::
COMM SFTON P0408
COMM MOVL C00462 BC00462 V=333.3
COMM MOVL C00463 BC00463 V=166.7
COMM MOVL C00464 BC00464 V=133.3 PL=0
COMM MACRO1 MJ#(0) ARGF24
COMM ARCON
COMM MOVL C00465 BC00465 V=7.5
COMM ARCOF
COMM MOVL C00466 BC00466 V=83.3
COMM SFTOF
COMM '------------------------
COMM 'W61.25
COMM '------------------------
COMM SFTON P0409
COMM MOVL C00467 BC00467 V=333.3
COMM MOVL C00468 BC00468 V=150.0
COMM MOVL C00469 BC00469 V=133.3 PL=0
COMM MACRO1 MJ#(0) ARGF24
COMM ARCON
COMM MOVL C00470 BC00470 V=7.5
COMM ARCOF
COMM MOVL C00471 BC00471 V=166.7
COMM SFTOF
COMM '::::::::::::::::::::::::
COMM '::::::::::::::::::::::::
COMM '::::::::::::::::::::::::
COMM '::::::::::::::::::::::::
COMM '::::::::::::::::::::::::
COMM MOVL C00472 BC00472 V=333.3
COMM MOVJ C00473 BC00473 VJ=50.00
COMM MOVJ C00474 BC00474 VJ=50.00
COMM MOVJ C00475 BC00475 VJ=50.00
COMM MOVJ C00476 BC00476 VJ=50.00
MOVJ C00477 BC00477 VJ=80.00
'------------------------
'W255A
MOVL C00478 BC00478 V=500.0
MOVL C00479 BC00479 V=333.3
SFTON P0361
MOVL C00480 BC00480 V=133.3 PL=0
MACRO1 MJ#(0) ARGF29
ARCON
SFTON P0362
MOVL C00481 BC00481 V=12.5
ARCOF
MOVL C00482 BC00482 V=250.0
SFTOF
MOVL C00483 BC00483 V=333.3
MOVL C00484 BC00484 V=333.3
MOVL C00485 BC00485 V=500.0
MOVJ C00486 BC00486 VJ=50.00
MOVJ C00487 BC00487 VJ=50.00
MOVJ C00488 BC00488 VJ=80.00
MOVJ C00489 BC00489 VJ=50.00
MOVJ C00490 BC00490 VJ=50.00
MOVL C00491 BC00491 V=333.3
'------------------------
'W31.28
'------------------------
SFTON P0310
MOVL C00492 BC00492 V=333.3
MOVL C00493 BC00493 V=333.3
MOVL C00494 BC00494 V=166.7
SFTON P0309
MOVL C00495 BC00495 V=500.0
MOVL C00496 BC00496 V=133.3 PL=0
ARCON
MOVL C00497 BC00497 V=11.7
ARCOF
MOVL C00498 BC00498 V=166.7
SFTOF
COMM MOVL C00499 BC00499 V=66.7 PL=0
COMM MACRO1 MJ#(0) ARGF24
COMM ARCON
COMM MOVL C00500 BC00500 V=8.3
COMM ARCOF
MOVL C00501 BC00501 V=250.0
SFTOF
'------------------------
'W31.30
'------------------------
SFTON P0311
MOVL C00502 BC00502 V=333.3
MOVL C00503 BC00503 V=133.3 PL=0
MACRO1 MJ#(0) ARGF30
ARCON
MOVL C00504 BC00504 V=11.7
ARCOF
MOVL C00505 BC00505 V=166.7
MOVL C00506 BC00506 V=333.3
SFTON P0310
MOVL C00507 BC00507 V=166.7
ARCON
MOVL C00508 BC00508 V=11.7
ARCOF
SFTOF
MOVL C00509 BC00509 V=166.7
MOVL C00510 BC00510 V=333.3
SFTOF
MOVL C00511 BC00511 V=500.0
MOVL C00512 BC00512 V=333.3
'::::::::::::::::::::::::
'::::::::::::::::::::::::
'::::::::::::::::::::::::
'::::::::::::::::::::::::
'::::::::::::::::::::::::
'::::::::::::::::::::::::
'::::::::::::::::::::::::
MOVJ C00513 BC00513 VJ=50.00 PL=0
COMM MOVJ C00514 BC00514 VJ=50.00
COMM MOVJ C00515 BC00515 VJ=50.00
COMM '::::::::::::::::::::::::::::::::
COMM '::::::::::::::::::::::::::::::::
COMM '------------------------
COMM 'W61.30
COMM '------------------------
COMM '::::::::::::::::::::::::::::::::
COMM '::::::::::::::::::::::::::::::::
COMM SFTON P0411
COMM MOVL C00516 BC00516 V=333.3
COMM MOVL C00517 BC00517 V=133.3 PL=0
COMM MACRO1 MJ#(0) ARGF24
COMM ARCON
COMM MOVL C00518 BC00518 V=7.5
COMM ARCOF
COMM MOVL C00519 BC00519 V=166.7
COMM SFTOF
COMM MOVL C00520 BC00520 V=500.0
COMM MOVJ C00521 BC00521 VJ=50.00
COMM MOVJ C00522 BC00522 VJ=50.00
COMM MOVJ C00523 BC00523 VJ=50.00
COMM MOVJ C00524 BC00524 VJ=80.00
COMM MOVJ C00525 BC00525 VJ=80.00
COMM '------------------------
COMM 'W256A
COMM '------------------------
MOVJ C00526 BC00526 VJ=80.00
MOVJ C00527 BC00527 VJ=80.00
SFTON P0358
MOVL C00528 BC00528 V=333.3
MOVL C00529 BC00529 V=250.0
MOVL C00530 BC00530 V=166.7 PL=0
MACRO1 MJ#(0) ARGF29
ARCON
SFTOF
SFTON P0357
MOVL C00531 BC00531 V=12.5
ARCOF
MOVL C00532 BC00532 V=333.3
SFTOF
MOVJ C00533 BC00533 VJ=50.00
MOVJ C00534 BC00534 VJ=50.00
MOVJ C00535 BC00535 VJ=80.00
CALL JOB:FRONT_WELD_90ST-2_4740
CALL JOB:MOVE_OUT_OF_TUNNEL
END
